PROGRAM MAIN
VAR
	fbCounter : FB_Counter;
	fbCounter2 : FB_Counter;
	
END_VAR

fbCounter.M_AddCounterValue();

fbCounter2.M_AddCounterValue();

END_PROGRAM

(* stored: Version 1.1.0.1, ProductVersion 3.1.4024.9
   POU MAIN: Id {f1943cf0-4542-4ac6-8c5d-d98559e49964}, SpecialFunc None *)
